{attribute 'GeneratedUsingTerminal: EK1100-0000-0018'}
{attribute addProperty BoxType "EK1100-0000-0018"}
{attribute addProperty Id "Beckhoff_ER5xxxEK1122Beckhoff_ER5xxxEK1122_4863E8E680"}
{attribute addProperty CRC "1151938078"}
{attribute addProperty Size "80"}
TYPE Beckhoff_ER5xxx_44A92E1E EXTENDS EK1100_1FC0878B :
STRUCT
	{attribute addProperty Name "Beckhoff_ER5xxxEK1122"}
	{attribute addProperty PreviousPort "Beckhoff ER5xxx : B"}
	Beckhoff_ER5xxxEK1122 : Beckhoff_ER5xxxEK1122_4863E8E6;
END_STRUCT
END_TYPE

(* stored: Version 1.2.0.0, ProductVersion 3.1.4024.9
   DUT Beckhoff_ER5xxx_44A92E1E: Id {b50d5844-e733-412e-b7aa-040af9f6fd41} *)
